// TIA Portal project "Enfriamiento Basculante" (V15)

(* hardware
DEVICE "S7-1200 station_1"  S7-1200 Station
   slot 0: "Rack_0"  S7-1200 Rack  Rack  V1.0
   slot 1: "PLC_1"  CPU 1214C DC/DC/DC  6ES7 214-1AG40-0XB0  V4.2
*)

// ===== PLC "PLC_1"  CPU 1214C DC/DC/DC =====

VAR_GLOBAL   // PLC tag table "Tabla de variables estándar"
   "Marcha" AT %I0.0 : Bool;
   "Paro" AT %I0.1 : Bool;
   "OL" AT %I0.2 : Bool;
   "C_Bomba" AT %Q0.0 : Bool;
   "Sistema_Listo" AT %M10.0 : Bool;
   "Tag_1" AT %M10.1 : Bool;
   "Tag_2" AT %M10.2 : Bool;
   "Tag_3" AT %Q0.1 : Bool;
   "Tag_4" AT %M0.2 : Bool;
   "Tag_5" AT %M0.1 : Bool;
END_VAR

// folder: System blocks/Program resources

DATA_BLOCK "T1"   // DB1
{ S7_Optimized_Access := 'TRUE' }
AUTHOR : Simatic
FAMILY : IEC
NAME : IEC_TMR
VERSION : 1.0
// stored: InstanceOfName IEC_TIMER
"IEC_TIMER"
BEGIN
END_DATA_BLOCK

DATA_BLOCK "T2"   // DB2
{ S7_Optimized_Access := 'TRUE' }
AUTHOR : Simatic
FAMILY : IEC
NAME : IEC_TMR
VERSION : 1.0
// stored: InstanceOfName IEC_TIMER
"IEC_TIMER"
BEGIN
END_DATA_BLOCK

DATA_BLOCK "TA"   // DB3
{ S7_Optimized_Access := 'TRUE' }
AUTHOR : Simatic
FAMILY : IEC
NAME : IEC_TMR
VERSION : 1.0
// stored: InstanceOfName IEC_TIMER
"IEC_TIMER"
BEGIN
END_DATA_BLOCK

DATA_BLOCK "TB"   // DB4
{ S7_Optimized_Access := 'TRUE' }
AUTHOR : Simatic
FAMILY : IEC
NAME : IEC_TMR
VERSION : 1.0
// stored: InstanceOfName IEC_TIMER
"IEC_TIMER"
BEGIN
END_DATA_BLOCK

// folder: (top level)

FUNCTION "Control de enfriamiento" : Void   // FC1, LAD
{ S7_Optimized_Access := 'TRUE' }
VERSION : 0.1
BEGIN

REGION Network 1
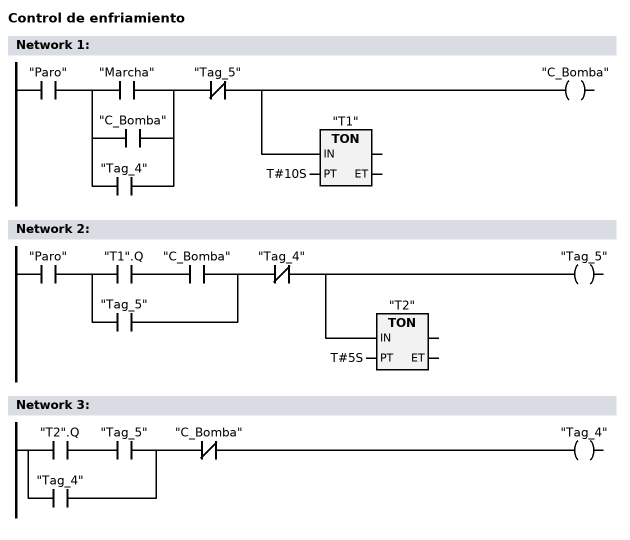
   "C_Bomba" := "Paro" AND ("Marcha" OR "C_Bomba" OR "Tag_4") AND NOT "Tag_5";
   "T1".TON(IN := "C_Bomba", PT := T#10S);
END_REGION

REGION Network 2
   "Tag_5" := "Paro" AND (("T1".Q AND "C_Bomba") OR "Tag_5") AND NOT "Tag_4";
   "T2".TON(IN := "Tag_5", PT := T#5S);
END_REGION

REGION Network 3
   RUNG wire#powerrail
      Contact( "T2".Q )
      Contact( "Tag_5" )
      wire#w1
      I_Contact( "C_Bomba" )
      Coil( "Tag_4" )
   END_RUNG
   RUNG wire#powerrail
      Contact( "Tag_4" )
   END_RUNG wire#w1
   // the same network as SCL:
   "Tag_4" := (("T2".Q AND "Tag_5") OR "Tag_4") AND NOT "C_Bomba";
END_REGION
END_FUNCTION

FUNCTION "Enfriamieno_SCL" : Void   // FC2, SCL
{ S7_Optimized_Access := 'TRUE' }
VERSION : 0.1
BEGIN
   IF "Marcha" THEN
       "Sistema_Listo" := 1; //set sisemas listo
   END_IF;

   IF NOT "Paro" THEN
       "Sistema_Listo" := 0; //reset sisemas listo
   END_IF;

   //Temporizadores
   //
   "TA".TON(IN:="Sistema_Listo" AND NOT "TB".Q,
            PT:=T#10s);

   "TB".TON(IN:="TA".Q,
            PT:=T#5s);

   "C_Bomba" := ("TA".Q AND NOT "TB".Q);
END_FUNCTION

ORGANIZATION_BLOCK "Main"   // OB1, LAD, ProgramCycle
TITLE = "Main Program Sweep (Cycle)"
{ S7_Optimized_Access := 'TRUE' }
VERSION : 0.1
   VAR_INPUT
      Initial_Call : Bool;   // Initial call of this OB
      Remanence : Bool;   // =True, if remanent data are available
   END_VAR
BEGIN

REGION Network 1
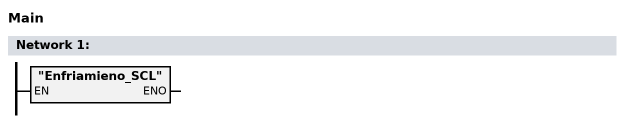
   RUNG wire#powerrail
      "Enfriamieno_SCL"()
   END_RUNG
   // the same network as SCL:
   "Enfriamieno_SCL"();
END_REGION
END_ORGANIZATION_BLOCK